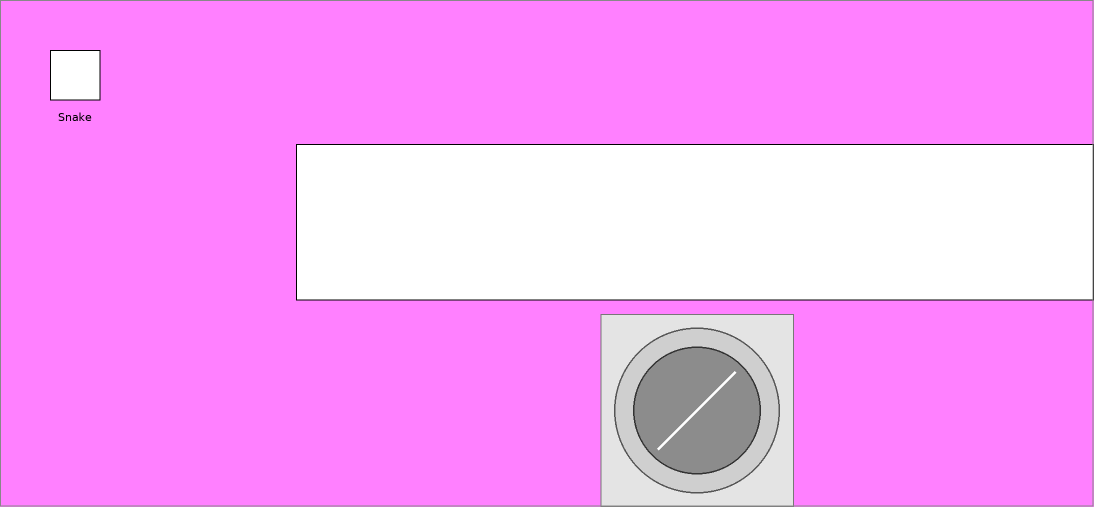
VISUALIZATION EkranGlowny  // 1094x507
    RoundedRectangle (50,50 50x50)
        p3560616238: MAIN.ObranPoczatkowy.iRuchX
        p2738717112: MAIN.ObranPoczatkowy.iRuchY
        OnMouseClick: change screen: Snake
    Rectangle (50,105 50x25), "Snake"
        p3560616238: MAIN.ObranPoczatkowy.iRuchX
        p2738717112: MAIN.ObranPoczatkowy.iRuchY
    Potentiometer360 (599,314 196x193), variable: MAIN.ObranPoczatkowy.predkoscRuchu, style: Potentiometer-Potentiometer360-Gray, scale format: %.1f, scale 1..111
        p2431819421: Outside
    RoundedRectangle (296,144 798x156), "Nalerzy kliknąć ikonkę żeby przejść dalej"
END_VISUALIZATION

(* stored: Version 1.1.0.1, ProductVersion 3.1.4024.4
   Visu EkranGlowny: Id {c1fe4e5c-65e9-46b6-ac15-b0ee5e746a3c} *)
